// TwinCAT 3 PLC project Sys1_PLC
// ProgramVersion: 3.1.4026.26
// libraries:
//   Tc2_Standard, * (Beckhoff Automation GmbH)
//   Tc2_System, * (Beckhoff Automation GmbH)
// project tree:
//   DUTs/ Auto_Test_DB_DUT.TcDUT (not stored), Auto_Test_DUT.TcDUT (not stored), Barcode_Station_DUT.TcDUT, Charger_DUT.TcDUT, Gate_Station_DUT.TcDUT (not stored), Level_Keys_DUT.TcDUT (not stored)
//   DUTs/Conveyors/ Buffer_Cnv_Control_DUT.TcDUT, Buffer_Cnv_Inputs_DUT.TcDUT (not stored), Buffer_Cnv_Settings_DUT.TcDUT (not stored), Cnv_Errors_DUT.TcDUT, Cnv_Inputs_DUT.TcDUT, Cnv_Instruction_DUT.TcDUT (not stored), Cnv_Level_Control_DUT.TcDUT (not stored), Cnv_Level_Inputs_DUT.TcDUT (not stored), Cnv_Level_Settings_DUT.TcDUT (not stored), Cnv_Motor_DUT.TcDUT, Cnv_VTD_Control_DUT.TcDUT, Cnv_VTD_Settings_DUT.TcDUT (not stored), ECnv_Control_DUT.TcDUT (not stored), ECnv_Settings_DUT.TcDUT (not stored)
//   DUTs/Safety_Stops/ Sfts_Control_DUT.TcDUT (not stored), Sfts_Inputs_DUT.TcDUT (not stored), Sfts_Instruction_DUT.TcDUT (not stored), Sfts_Settings_DUT.TcDUT (not stored)
//   DUTs/System/ ID_Decoded_DUT.TcDUT (not stored), OrderTable_DUT.TcDUT (not stored), System_DUT.TcDUT (not stored), System_Settings_DUT.TcDUT, WMS_OPC_UA_DUT.TcDUT
//   DUTs/VTD/ VTD_Control_DUT.TcDUT, VTD_Errors_DUT.TcDUT (not stored), VTD_Inputs_DUT.TcDUT (not stored), VTD_Instruction_DUT.TcDUT (not stored), VTD_Levels_DUT.TcDUT (not stored), VTD_Motor_DUT.TcDUT (not stored), VTD_Outputs_DUT.TcDUT (not stored), VTD_Settings_DUT.TcDUT (not stored), VTD_Shuttle_Interlock_DUT.TcDUT
//   GVLs/ Bypass.TcGVL, CNV_HMI_IO.TcGVL (not stored), Control.TcGVL (not stored), Errors.TcGVL (not stored), Force.TcGVL, Settings.TcGVL (not stored), System_Control.TcGVL
//   GVLs/HMI/ CNV_HMI.TcGVL (not stored)
//   GVLs/IO/ IO_Panel.TcGVL (not stored)
//   / PlcTask.TcTTO (not stored)
//   POUs/Conveyors/ Buffer_Conveyor_FB.TcPOU (not stored)
//   POUs/ MAIN.TcPOU, Stack_Lights_FB.TcPOU (not stored)
//   POUs/System/ Conveyors_Transfer.TcPOU (not stored)
//   POUs/System/Functions/ ID_Decode_F.TcPOU, Set_Bit_F.TcPOU (not stored)
//   POUs/VTD/ Light_Bars_FB.TcPOU (not stored), VTD_FB.TcPOU (not stored)
// real-time tasks:
//   TASK PlcTask: cycle T#10ms, priority 20, ADS port 350
// I/O:
//   DEVICE VTD_1 (EtherCAT), AmsNetId 192.168.0.103.2.1
//     DI-01 (EPP1008-0022) [EPP1008-0022 8 Ch. Dig. Input 24V, 3ms, M12]
//     DI-02 (EPP1008-0022) [EPP1008-0022 8 Ch. Dig. Input 24V, 3ms, M12]
//     DI-03 (EPP1008-0022) [EPP1008-0022 8 Ch. Dig. Input 24V, 3ms, M12]
//     DI-04 (EPP1008-0022) [EPP1008-0022 8 Ch. Dig. Input 24V, 3ms, M12]
//     DI-05 (EPP1008-0022) [EPP1008-0022 8 Ch. Dig. Input 24V, 3ms, M12]
//     DI-06 (EPP1008-0022) [EPP1008-0022 8 Ch. Dig. Input 24V, 3ms, M12]
//     DI-07 (EPP1008-0022) [EPP1008-0022 8 Ch. Dig. Input 24V, 3ms, M12]
//     DI-08 (EPP1008-0022) [EPP1008-0022 8 Ch. Dig. Input 24V, 3ms, M12]
//     DI-09 (EPP1008-0022) [EPP1008-0022 8 Ch. Dig. Input 24V, 3ms, M12]
//     DI-10 (EPP1008-0022) [EPP1008-0022 8 Ch. Dig. Input 24V, 3ms, M12]
//     ENCODER (EPP5001-0002) [EPP5001-0002 1Ch. SSI Encoder]
//     DIO-01 (EPP2328-0002) [EPP2328-0002 4 CH. Dig. In, 3ms, 4 Ch. Dig. Out 24V, 2A, M12]
//     DIO-02 (EPP2328-0002) [EPP2328-0002 4 CH. Dig. In, 3ms, 4 Ch. Dig. Out 24V, 2A, M12]
//     DIO-03 (EPP2328-0002) [EPP2328-0002 4 CH. Dig. In, 3ms, 4 Ch. Dig. Out 24V, 2A, M12]
//     DIO-04 (EPP2328-0002) [EPP2328-0002 4 CH. Dig. In, 3ms, 4 Ch. Dig. Out 24V, 2A, M12]
//     DIO-05 (EPP2328-0002) [EPP2328-0002 4 CH. Dig. In, 3ms, 4 Ch. Dig. Out 24V, 2A, M12]
//     DIO-06 (EPP2328-0002) [EPP2328-0002 4 CH. Dig. In, 3ms, 4 Ch. Dig. Out 24V, 2A, M12]
//     DIO-07 (EPP2328-0002) [EPP2328-0002 4 CH. Dig. In, 3ms, 4 Ch. Dig. Out 24V, 2A, M12]
//     DI-11 (EPP1809-0022) [EPP1809-0022 16 Ch. Dig. Input 24V, 3ms, M8]
//     FDI-01 (EP1918-0002) [EP1918, 8Ch. Safety Input 24V, TwinSAFE]
//       modules: Module 1 (FSOE), Module 2 (FSLOGIC)
//     PLC_CONTROLLER (EK1200) [EK1200-5000 EtherCAT Power supply (2A E-Bus)]
//       DI-01 (EL1809) [EL1809 16Ch. Dig. Input 24V, 3ms]
//       DI-02 (EL1809) [EL1809 16Ch. Dig. Input 24V, 3ms]
//       DO-01 (EL2809) [EL2809 16Ch. Dig. Output 24V, 0.5A]
//       DO-02 (EL2809) [EL2809 16Ch. Dig. Output 24V, 0.5A]
//       F-PLC (EL6910) [EL6910, TwinSAFE PLC]
//       FDI-01 (EL1918) [EL1918, 8Ch. Safety Input 24V, TwinSAFE]
//         modules: Module 1 (FSOE), Module 2 (FSLOGIC)
//       FDO-01 (EL2912) [EL2912, 2Ch. Safety Output 24V, 2A, TwinSAFE]
//         modules: Module 1 (FSOE), Module 2 (FSOUT), Module 3 (DEVICEIO), Module 4 (FSLOGIC)
//       ETHERCAT-1 (EK1322) [EK1322 2-port EtherCAT P junction with feed-in]
//       ETHERCAT-2 (EK1322) [EK1322 2-port EtherCAT P junction with feed-in]
//       ETHERCAT-3 (EK1322) [EK1322 2-port EtherCAT P junction with feed-in]
//       PROFNET (EL6633) [EL6633 PROFINET IO Controller]
//       ETHERCAT-4 (EK1122) [EK1122 2 port EtherCAT junction]
//       POWER_SUPPLY (EL9410) [EL9410 E-Bus Power Supplier  (Diagnostics)]
//       END_TERMINAL (EL9011) [EL9011 End Terminal]
//   DEVICE MAIN (EtherCAT), AmsNetId 192.168.0.103.3.1
//     Term 36 (EK1200) [EK1200-5000 EtherCAT Power supply (2A E-Bus)]
//       DI-01 (EL1809) [EL1809 16Ch. Dig. Input 24V, 3ms]
//       DI-02 (EL1809) [EL1809 16Ch. Dig. Input 24V, 3ms]
//       DO-01 (EL2809) [EL2809 16Ch. Dig. Output 24V, 0.5A]
//       DO-02 (EL2809) [EL2809 16Ch. Dig. Output 24V, 0.5A]
//       F-PLC (EL6910) [EL6910, TwinSAFE PLC]
//       FDI-01 (EL1918) [EL1918, 8Ch. Safety Input 24V, TwinSAFE]
//         modules: Module 1 (FSOE), Module 2 (FSLOGIC)
//       FDI-02 (EL1918) [EL1918, 8Ch. Safety Input 24V, TwinSAFE]
//         modules: Module 1 (FSOE), Module 2 (FSLOGIC)
//       FDO-01 (EL2912) [EL2912, 2Ch. Safety Output 24V, 2A, TwinSAFE]
//         modules: Module 1 (FSOE), Module 2 (FSOUT), Module 3 (DEVICEIO), Module 4 (FSLOGIC)
//       FDO-02 (EL2912) [EL2912, 2Ch. Safety Output 24V, 2A, TwinSAFE]
//         modules: Module 1 (FSOE), Module 2 (FSOUT), Module 3 (DEVICEIO), Module 4 (FSLOGIC)
//       POWER_SUPPLY (EL9410) [EL9410 E-Bus Power Supplier  (Diagnostics)]
//       PROFNET (EL6633) [EL6633 PROFINET IO Controller]
//       ETHERCAT (EK1322) [EK1322 2-port EtherCAT P junction with feed-in]
//       END_TERMINAL (EL9011) [EL9011 End Terminal]

// ---- DUTs/Barcode_Station_DUT.TcDUT
TYPE Barcode_Station_DUT :
STRUCT
	Start:	BOOL;
	Ready:	BOOL;
	Running:	BOOL;
	Done:	BOOL;
	Valid:	BOOL;
	Reading_Gate_number:	STRING;
	Reading_Gate_number_OLD:	STRING;
	Number_OF_Reading_Gates:	STRING;
	Number_OF_Reading_Gates_OLD:	STRING;
	Barcode:	STRING;
	Barcode_Old:	STRING;
END_STRUCT
END_TYPE

// ---- DUTs/Charger_DUT.TcDUT
TYPE Charger_DUT :
STRUCT
	Output_Voltage:	REAL;                   	//Actual Output Voltage  
	Output_Current:	REAL;                       //Actual Output Current  
	Set_Voltage_Feedback:	REAL;               //Set Voltage Value      
	Set_Current_Feedback:	REAL;               //Set Current Value      
	Charging_Start:	BOOL;                       //Charging Running Status
	Set_Voltage_Output:	REAL;                   //Issue Target Voltage   
	Set_Current_Output:	REAL;                   //Issue Target Current   
	Start_Charging:	BOOL;                       //Start Charging Command 
	Stop_Charging:	BOOL;                       //Stop Charging Command  
	Confirm_Voltage_Current_Setting:	BOOL;   //Confirmation Command   
END_STRUCT
END_TYPE

// ---- DUTs/Conveyors/Buffer_Cnv_Control_DUT.TcDUT
TYPE Buffer_Cnv_Control_DUT :
STRUCT
	Mode:	UINT;
	Error:	BOOL;
	Warning:	UINT;
	Enabled:	BOOL;
	Stopped:	BOOL;
	Done:	BOOL;
	Running:	BOOL;
	Ready_For_Task:	BOOL;
	Current_Task_Type:	UINT;
	Current_Task_ID:	UINT;
	Cnv_Occupied:	BOOL;
	SM_State:	UINT;
	Motor:	Cnv_Motor_DUT;
	Instruction:	Cnv_Instruction_DUT;
	Inputs:	Buffer_Cnv_Inputs_DUT;
	Safety_Stop_Cnrl:	Sfts_Control_DUT;
	Cnv_Errors:	Cnv_Errors_DUT;
END_STRUCT
END_TYPE

// ---- DUTs/Conveyors/Cnv_Errors_DUT.TcDUT
TYPE Cnv_Errors_DUT :
STRUCT
	Error_Word_1:	UINT;
	Error_Word_2:	UINT;
	Error_Word_3:	UINT;
	Error_Word_4:	UINT;
END_STRUCT
END_TYPE

// ---- DUTs/Conveyors/Cnv_Inputs_DUT.TcDUT
TYPE Cnv_Inputs_DUT :
STRUCT
	Forward_Sensor:	BOOL;
	Backward_Sensor:	BOOL;
	VFD_Status:	WORD;
	VFD_Speed_Actual:	INT;
	VFD_ActualCurrent:	INT;
	VFD_ActualTorque:	INT;
END_STRUCT
END_TYPE

// ---- DUTs/Conveyors/Cnv_Motor_DUT.TcDUT
TYPE Cnv_Motor_DUT :
STRUCT
	Enable:	BOOL;
	Enabled:	BOOL;
	Ready:	BOOL;
	Forward:	BOOL;
	Reverse:	BOOL;
	Speed:	REAL;
	Speed_Actual:	REAL;
	Actual_Current:	REAL;
	Actual_Torque:	UINT;
	Config_Axis:	WORD;
	Error:	BOOL;
	Status:	WORD;
	Communication_Error:	WORD;
	Lockout:	BOOL;
END_STRUCT
END_TYPE

// ---- DUTs/Conveyors/Cnv_VTD_Control_DUT.TcDUT
TYPE Cnv_VTD_Control_DUT :
STRUCT
	Cnv_Level:	ARRAY[2..6] OF Cnv_Level_Control_DUT;
END_STRUCT
END_TYPE

// ---- DUTs/System/System_Settings_DUT.TcDUT
TYPE System_Settings_DUT :
STRUCT
	VTD_Count:  UINT;
	Level_Count:  UINT;
	Cnv_Count:  UInt;
	Shuttle_Count:  UInt;
	Shuttle_Interlock_Timeout:  UINT;
END_STRUCT
END_TYPE

// ---- DUTs/System/WMS_OPC_UA_DUT.TcDUT
TYPE WMS_OPC_UA_DUT :
STRUCT
	Task_ID:  INT;
	Task_Metadata:  STRING[250];
	Task_Type:  Int;
	Source_Location:  DInt;
	Destination_Location:  DInt;
	Task_Data_Available:  Bool;
	SM_State:  UInt;
	Movement_Ready:  Bool;
	Movement_Request_Complete:  Bool;
	Movement_Request_Complete_Ack:  Bool;
	Shuttle_ID:  Int;
	Shuttle_Loaded:  Bool;
	Pallet_Type:  BYTE;
	Pallet_Alignment:  BYTE;
	SM_State_Maestro:  UInt;
	Pallet_Weight:  INT;
END_STRUCT
END_TYPE

// ---- DUTs/VTD/VTD_Control_DUT.TcDUT
TYPE VTD_Control_DUT :
STRUCT
	Mode:	UINT;
	Error:	BOOL;
	Warning:	UINT;
	Enabled:	BOOL;
	Stopped:	BOOL;
	Running:	BOOL;
	Done:	BOOL;
	Current_Task_Type:	UINT;
	Current_Task_ID:	UINT;
	AbsoluteEnc:	REAL;
	LinearEnc:	REAL;
	Current_Level:	UINT;
	Docked:	BOOL;
	LP_State:	UINT;
	DP_Extended:	BOOL;
	Pallet_Loaded:	UINT;
	Shuttle_Loaded:	UINT;
	SM_State:	UINT;
	Motor_UP:	BOOL;
	Motor_Down:	BOOL;
	Motor_Speed:	UINT;
	VFD_Error:	UINT;
	LE_Error:	UINT;
	AE_Error:	UINT;
	Encoder_Delta:	INT;
	Instruction:	VTD_Instruction_DUT;
	Shuttle_Interlock:	VTD_Shuttle_Interlock_DUT;
	Inputs:	VTD_Inputs_DUT;
	Outputs:	VTD_Outputs_DUT;
	Motor:	VTD_Motor_DUT;
	VTD_Errors:	VTD_Errors_DUT;
END_STRUCT
END_TYPE

// ---- DUTs/VTD/VTD_Shuttle_Interlock_DUT.TcDUT
TYPE VTD_Shuttle_Interlock_DUT :
STRUCT
	Interlock_Complete:  BOOL;
	Interlock_Complete_Ack:  BOOL;
	Ready_To_Interlock:  Bool;
	Interlock_Request:  Bool;
	Shuttle_ID:  UInt;
	Shuttle_Target_Location:  DInt;
	Shuttle_Start_Location:  DInt;
	Shuttle_Loaded:  Bool;
	Shuttle_Interlock_Task_ID:  UInt;
	Shuttle_Interlock_Task_Metadata:  STRING;
END_STRUCT
END_TYPE

// ---- GVLs/Bypass.TcGVL
{attribute 'qualified_only'}
VAR_GLOBAL
	Remote_Panel_1:  Safety_Bypass_RemotePanel;
	Remote_Panel_2:  Safety_Bypass_RemotePanel;
END_VAR

// ---- GVLs/Force.TcGVL
{attribute 'qualified_only'}
VAR_GLOBAL
	Remote_Panel:  ARRAY[1..2] OF STRUCT;
END_VAR

// ---- GVLs/System_Control.TcGVL
{attribute 'qualified_only'}
VAR_GLOBAL
	Reset_All:  BOOL;
	MQTT_Enable:  BOOL;
	OPC_Enable:  Bool;
END_VAR

// ---- POUs/MAIN.TcPOU
PROGRAM MAIN
VAR
	VTD : VTD_FB;
END_VAR

VTD.

END_PROGRAM

// ---- POUs/System/Functions/ID_Decode_F.TcPOU
FUNCTION ID_Decode_F : BOOL
VAR_INPUT
	ID: DINT;
END_VAR
VAR_IN_OUT
	ID_Decoded: ID_Decoded_DUT;
END_VAR
VAR
END_VAR

// Extract XX (first two digits)
ID_Decoded.Device_Type := DINT_TO_INT(ID / 10000);        // 123456 / 10000 = 12

// Extract YY (middle two digits)
ID_Decoded.Level := DINT_TO_INT((ID MOD 10000) / 100); // 123456 % 10000 = 3456 → 3456 / 100 = 34

// Extract ZZ (last two digits)
ID_Decoded.VTD := DINT_TO_INT(ID MOD 100);       // 123456 % 100 = 56

END_FUNCTION
